FUNCTION F_IncIndex : INT
VAR_INPUT
	IDX:	INT;		// Index to be incremented
	IdxMIN:	INT;		// Min Value for index	
	IdxMAX:	INT;		// Max Value for index
END_VAR
VAR
END_VAR

IF IDX < IdxMAX THEN
	F_IncIndex := IDX + 1; 
ELSIF IDX = IdxMAX THEN
	F_IncIndex := IdxMIN;
ELSIF IDX < IdxMIN OR IDX > IdxMAX THEN
	F_IncIndex := IdxMIN;
END_IF

END_FUNCTION

(* stored: Version 1.1.0.1, ProductVersion 3.1.4024.4
   POU F_IncIndex: Id {ea33e8f4-f842-4a2a-a6c2-b0e11b61b6f3}, SpecialFunc None *)
